{attribute addProperty BoxType "APS4322-7000-0017"}
{attribute addProperty Id "ControlWordAT %Q*UINT16217Current_D_0X0AT %Q*INT1622Current_D_0X1AT %Q*INT1623Current_D_0X2AT %Q*INT1624Current_D_0Y0AT %Q*INT1625Current_D_0Y1AT %Q*INT1626Current_D_0Y2AT %Q*INT1627Current_D_1X0AT %Q*INT1628Current_D_1X1AT %Q*INT1629Current_D_1X2AT %Q*INT16210Current_D_1Y0AT %Q*INT16211Current_D_1Y1AT %Q*INT16212Current_D_1Y2AT %Q*INT16213Current_D_2X0AT %Q*INT16214Current_D_2X1AT %Q*INT16215Current_D_2X2AT %Q*INT16216Current_D_2Y0AT %Q*INT16217Current_D_2Y1AT %Q*INT16218Current_D_2Y2AT %Q*INT16219Current_D_3X0AT %Q*INT16220Current_D_3X1AT %Q*INT16221Current_D_3X2AT %Q*INT16222Current_D_3Y0AT %Q*INT16223Current_D_3Y1AT %Q*INT16224Current_D_3Y2AT %Q*INT16225Current_Q_0X0AT %Q*INT16226Current_Q_0X1AT %Q*INT16227Current_Q_0X2AT %Q*INT16228Current_Q_0Y0AT %Q*INT16229Current_Q_0Y1AT %Q*INT16230Current_Q_0Y2AT %Q*INT16231Current_Q_1X0AT %Q*INT16232Current_Q_1X1AT %Q*INT16233Current_Q_1X2AT %Q*INT16234Current_Q_1Y0AT %Q*INT16235Current_Q_1Y1AT %Q*INT16236Current_Q_1Y2AT %Q*INT16237Current_Q_2X0AT %Q*INT16238Current_Q_2X1AT %Q*INT16239Current_Q_2X2AT %Q*INT16240Current_Q_2Y0AT %Q*INT16241Current_Q_2Y1AT %Q*INT16242Current_Q_2Y2AT %Q*INT16243Current_Q_3X0AT %Q*INT16244Current_Q_3X1AT %Q*INT16245Current_Q_3X2AT %Q*INT16246Current_Q_3Y0AT %Q*INT16247Current_Q_3Y1AT %Q*INT16248Current_Q_3Y2AT %Q*INT16249PhiE_0X0AT %Q*UINT16250PhiE_0X1AT %Q*UINT16251PhiE_0X2AT %Q*UINT16252PhiE_0Y0AT %Q*UINT16253PhiE_0Y1AT %Q*UINT16254PhiE_0Y2AT %Q*UINT16255PhiE_1X0AT %Q*UINT16256PhiE_1X1AT %Q*UINT16257PhiE_1X2AT %Q*UINT16258PhiE_1Y0AT %Q*UINT16259PhiE_1Y1AT %Q*UINT16260PhiE_1Y2AT %Q*UINT16261PhiE_2X0AT %Q*UINT16262PhiE_2X1AT %Q*UINT16263PhiE_2X2AT %Q*UINT16264PhiE_2Y0AT %Q*UINT16265PhiE_2Y1AT %Q*UINT16266PhiE_2Y2AT %Q*UINT16267PhiE_3X0AT %Q*UINT16268PhiE_3X1AT %Q*UINT16269PhiE_3X2AT %Q*UINT16270PhiE_3Y0AT %Q*UINT16271PhiE_3Y1AT %Q*UINT16272PhiE_3Y2AT %Q*UINT16273"}
{attribute addProperty CRC "215048737"}
{attribute addProperty SizeInBites "1168"}
{attribute addProperty SizeInBytes "146"}
TYPE APS_Outputs_0CD16221 :
STRUCT
	{attribute addProperty Name "ControlWord"}
	ControlWord AT %Q* : UINT;
	{attribute addProperty Name "Current_D_0X0"}
	Current_D_0X0 AT %Q* : INT;
	{attribute addProperty Name "Current_D_0X1"}
	Current_D_0X1 AT %Q* : INT;
	{attribute addProperty Name "Current_D_0X2"}
	Current_D_0X2 AT %Q* : INT;
	{attribute addProperty Name "Current_D_0Y0"}
	Current_D_0Y0 AT %Q* : INT;
	{attribute addProperty Name "Current_D_0Y1"}
	Current_D_0Y1 AT %Q* : INT;
	{attribute addProperty Name "Current_D_0Y2"}
	Current_D_0Y2 AT %Q* : INT;
	{attribute addProperty Name "Current_D_1X0"}
	Current_D_1X0 AT %Q* : INT;
	{attribute addProperty Name "Current_D_1X1"}
	Current_D_1X1 AT %Q* : INT;
	{attribute addProperty Name "Current_D_1X2"}
	Current_D_1X2 AT %Q* : INT;
	{attribute addProperty Name "Current_D_1Y0"}
	Current_D_1Y0 AT %Q* : INT;
	{attribute addProperty Name "Current_D_1Y1"}
	Current_D_1Y1 AT %Q* : INT;
	{attribute addProperty Name "Current_D_1Y2"}
	Current_D_1Y2 AT %Q* : INT;
	{attribute addProperty Name "Current_D_2X0"}
	Current_D_2X0 AT %Q* : INT;
	{attribute addProperty Name "Current_D_2X1"}
	Current_D_2X1 AT %Q* : INT;
	{attribute addProperty Name "Current_D_2X2"}
	Current_D_2X2 AT %Q* : INT;
	{attribute addProperty Name "Current_D_2Y0"}
	Current_D_2Y0 AT %Q* : INT;
	{attribute addProperty Name "Current_D_2Y1"}
	Current_D_2Y1 AT %Q* : INT;
	{attribute addProperty Name "Current_D_2Y2"}
	Current_D_2Y2 AT %Q* : INT;
	{attribute addProperty Name "Current_D_3X0"}
	Current_D_3X0 AT %Q* : INT;
	{attribute addProperty Name "Current_D_3X1"}
	Current_D_3X1 AT %Q* : INT;
	{attribute addProperty Name "Current_D_3X2"}
	Current_D_3X2 AT %Q* : INT;
	{attribute addProperty Name "Current_D_3Y0"}
	Current_D_3Y0 AT %Q* : INT;
	{attribute addProperty Name "Current_D_3Y1"}
	Current_D_3Y1 AT %Q* : INT;
	{attribute addProperty Name "Current_D_3Y2"}
	Current_D_3Y2 AT %Q* : INT;
	{attribute addProperty Name "Current_Q_0X0"}
	Current_Q_0X0 AT %Q* : INT;
	{attribute addProperty Name "Current_Q_0X1"}
	Current_Q_0X1 AT %Q* : INT;
	{attribute addProperty Name "Current_Q_0X2"}
	Current_Q_0X2 AT %Q* : INT;
	{attribute addProperty Name "Current_Q_0Y0"}
	Current_Q_0Y0 AT %Q* : INT;
	{attribute addProperty Name "Current_Q_0Y1"}
	Current_Q_0Y1 AT %Q* : INT;
	{attribute addProperty Name "Current_Q_0Y2"}
	Current_Q_0Y2 AT %Q* : INT;
	{attribute addProperty Name "Current_Q_1X0"}
	Current_Q_1X0 AT %Q* : INT;
	{attribute addProperty Name "Current_Q_1X1"}
	Current_Q_1X1 AT %Q* : INT;
	{attribute addProperty Name "Current_Q_1X2"}
	Current_Q_1X2 AT %Q* : INT;
	{attribute addProperty Name "Current_Q_1Y0"}
	Current_Q_1Y0 AT %Q* : INT;
	{attribute addProperty Name "Current_Q_1Y1"}
	Current_Q_1Y1 AT %Q* : INT;
	{attribute addProperty Name "Current_Q_1Y2"}
	Current_Q_1Y2 AT %Q* : INT;
	{attribute addProperty Name "Current_Q_2X0"}
	Current_Q_2X0 AT %Q* : INT;
	{attribute addProperty Name "Current_Q_2X1"}
	Current_Q_2X1 AT %Q* : INT;
	{attribute addProperty Name "Current_Q_2X2"}
	Current_Q_2X2 AT %Q* : INT;
	{attribute addProperty Name "Current_Q_2Y0"}
	Current_Q_2Y0 AT %Q* : INT;
	{attribute addProperty Name "Current_Q_2Y1"}
	Current_Q_2Y1 AT %Q* : INT;
	{attribute addProperty Name "Current_Q_2Y2"}
	Current_Q_2Y2 AT %Q* : INT;
	{attribute addProperty Name "Current_Q_3X0"}
	Current_Q_3X0 AT %Q* : INT;
	{attribute addProperty Name "Current_Q_3X1"}
	Current_Q_3X1 AT %Q* : INT;
	{attribute addProperty Name "Current_Q_3X2"}
	Current_Q_3X2 AT %Q* : INT;
	{attribute addProperty Name "Current_Q_3Y0"}
	Current_Q_3Y0 AT %Q* : INT;
	{attribute addProperty Name "Current_Q_3Y1"}
	Current_Q_3Y1 AT %Q* : INT;
	{attribute addProperty Name "Current_Q_3Y2"}
	Current_Q_3Y2 AT %Q* : INT;
	{attribute addProperty Name "PhiE_0X0"}
	PhiE_0X0 AT %Q* : UINT;
	{attribute addProperty Name "PhiE_0X1"}
	PhiE_0X1 AT %Q* : UINT;
	{attribute addProperty Name "PhiE_0X2"}
	PhiE_0X2 AT %Q* : UINT;
	{attribute addProperty Name "PhiE_0Y0"}
	PhiE_0Y0 AT %Q* : UINT;
	{attribute addProperty Name "PhiE_0Y1"}
	PhiE_0Y1 AT %Q* : UINT;
	{attribute addProperty Name "PhiE_0Y2"}
	PhiE_0Y2 AT %Q* : UINT;
	{attribute addProperty Name "PhiE_1X0"}
	PhiE_1X0 AT %Q* : UINT;
	{attribute addProperty Name "PhiE_1X1"}
	PhiE_1X1 AT %Q* : UINT;
	{attribute addProperty Name "PhiE_1X2"}
	PhiE_1X2 AT %Q* : UINT;
	{attribute addProperty Name "PhiE_1Y0"}
	PhiE_1Y0 AT %Q* : UINT;
	{attribute addProperty Name "PhiE_1Y1"}
	PhiE_1Y1 AT %Q* : UINT;
	{attribute addProperty Name "PhiE_1Y2"}
	PhiE_1Y2 AT %Q* : UINT;
	{attribute addProperty Name "PhiE_2X0"}
	PhiE_2X0 AT %Q* : UINT;
	{attribute addProperty Name "PhiE_2X1"}
	PhiE_2X1 AT %Q* : UINT;
	{attribute addProperty Name "PhiE_2X2"}
	PhiE_2X2 AT %Q* : UINT;
	{attribute addProperty Name "PhiE_2Y0"}
	PhiE_2Y0 AT %Q* : UINT;
	{attribute addProperty Name "PhiE_2Y1"}
	PhiE_2Y1 AT %Q* : UINT;
	{attribute addProperty Name "PhiE_2Y2"}
	PhiE_2Y2 AT %Q* : UINT;
	{attribute addProperty Name "PhiE_3X0"}
	PhiE_3X0 AT %Q* : UINT;
	{attribute addProperty Name "PhiE_3X1"}
	PhiE_3X1 AT %Q* : UINT;
	{attribute addProperty Name "PhiE_3X2"}
	PhiE_3X2 AT %Q* : UINT;
	{attribute addProperty Name "PhiE_3Y0"}
	PhiE_3Y0 AT %Q* : UINT;
	{attribute addProperty Name "PhiE_3Y1"}
	PhiE_3Y1 AT %Q* : UINT;
	{attribute addProperty Name "PhiE_3Y2"}
	PhiE_3Y2 AT %Q* : UINT;
END_STRUCT
END_TYPE

(* stored: Version 1.2.0.0, ProductVersion 3.1.4024.9
   DUT APS_Outputs_0CD16221: Id {11fb6284-53d5-4353-9f2d-bb7b3b64e1c2} *)
